(* CODESYS project Builder_Application_2RPi.project

Project tree, tasks and I/O mapping:
  Device : CODESYS Control for Raspberry Pi SL, 3S - Smart Software Solutions GmbH, version 3.5.11.0
    application Application
      libraries: Standard, * (System)
      task MainTask (cyclic, interval t#20ms, priority 1) calls PLC_PRG
      task VISU_TASK (cyclic, interval 100 ms, priority 31) calls VisuElems.Visu_Prg
      program PLC_PRG [ST]
      interface ITF_Builder: Set_Part1, Set_Part2, Set_Part3, Set_Main_Part
      function block ConcreteBuilder [ST]: Set_Main_Part, Set_Part1, Set_Part2, Set_Part3, Get_Main_Part, Get_Part1, Get_Part2, Get_Part3, Get_Result
      function block Director [ST]: fb_init, Construct
      function block Product [ST]: toString
      visualisation Visualization
    SoftMotion General Axis Pool
    GPIOs_A_B : GPIOs B+/Pi2, 3S - Smart Software Solutions GmbH, version 3.5.11.0
        unmapped channels: digital inputs (GPIO0..GPIO31), digital outputs (GPIO0..GPIO31)
    I²C
    SPI
    Onewire
    Camera device
      <Empty>
  libraries: VisuSymbols, 3.5.10.0 (System)
  text list GlobalTextList
*)

// Device/Application/PLC_PRG
PROGRAM PLC_PRG
VAR
	//Arrays with the different specifications for the Client to choose
	arrayChassis : ARRAY [1..3] OF STRING := ['Red Chassis ', 'Black Chassis ', 'White Chassis '];
	arrayCarType : ARRAY [1..3] OF STRING := ['Sedan ', 'Hatchback ', 'Sport '];
	arrayMotor : ARRAY [1..3] OF STRING := ['Motor 1.4cc ', 'Motor 2.0cc ', 'Motor 2.5cc '];
	arrayTires : ARRAY [1..3] OF STRING := ['Aluminium tires ', 'Chrome plated tires ', 'Ligth aluminium tires '];
	
	//Temporary array to have a reference to the clients choice
	tempArray : ARRAY [1..4] OF STRING;
	
	//Boolean and integer values to receive data from the tables in the visualization element
	//The boolean value validates if the client has chosen a valid option
	bChassis : BOOL := FALSE;
	//The integer value hold the reference to the array of specifications
	iChassis : INT := 0;
	
	//Boolean and integer values to receive data from the tables in the visualization element
	//The boolean value validates if the client has chosen a valid option
	bCarType : BOOL := FALSE;
	//The integer value hold the reference to the array of specifications
	iCarType : INT := 0;
	
	//Boolean and integer values to receive data from the tables in the visualization element
	//The boolean value validates if the client has chosen a valid option
	bMotor : BOOL := FALSE;
	//The integer value hold the reference to the array of specifications
	iMotor : INT := 0;
	
	//Boolean and integer values to receive data from the tables in the visualization element
	//The boolean value validates if the client has chosen a valid option
	bTires : BOOL := FALSE;
	//The integer value hold the reference to the array of specifications
	iTires : INT := 0;
	
	//Boolean value to verify and respond to a client's request
	bRequest : BOOL := FALSE;
	
	//String variable to interact and respond to the client in the visualization element
	sMessageLog : STRING := 'Waiting for your request';
	
	//A pointer to Poduct to dynamically create and delete product objects at the clients requests
	prod 	: POINTER TO Product;

	//A ConcreteBuilder instance to be passed to the Director and build the final Product objects
	aConcreteBuilder : ConcreteBuilder;
	
	//A Director instance that is instanciated with a ConcreteBuilder instance and the first specifications.
	// later on in the program these specifications of the ConcreteBuilder instance will be changed dynamically
	aDirector : Director(concreteBuilder:= aConcreteBuilder , specifications := tempArray);
	
END_VAR

//The visualization element has 4 coloums in which the client must select an option from each coloum.
//Once the client has made its choice, He can then procede to validate its request.
//The bottom rectangle will handle all possible responses from the application to the client.

//If the client makes a request in the visualization element
IF bRequest
	THEN
	//We verify that the cliet has chosen all the required parts(All in this case)
	IF bChassis AND bCarType AND bMotor AND bTires
		THEN
		//If the client has sent a valir request, the builder notifies the client about the received request
		sMessageLog := 'Your red car is being built';
		//A new product object is created on demand
		prod := __NEW(Product);
		//The tempArray is modified to the special characteristics demanded from the client on the visualization element
		tempArray[1] := arrayChassis[iChassis];
		tempArray[2] := arrayCarType[iCarType];
		tempArray[3] := arrayMotor[iMotor];
		tempArray[4] := arrayTires[iTires];

		//The Director object receives the specifications for the new Product to be built
		aDirector(spected := tempArray);
		//The Product object request the construction to the Director.
		prod^ := aDirector.Construct();
		//The Builder's response after the Director object has handled the proper request
		sMessageLog := CONCAT( 'Your car has been built. It has: ', prod^.toString());
		//Once this reques has been handled, the request flag is set to FALSE
		bRequest := FALSE;
		//Once this reques has been handled, the Product object is deleted to free memory
		__DELETE(prod);
		
		//If the client did not choose all the required parts
		ELSE
			
		//The Builder responds
		sMessageLog := 'You need to select all the parts for your car';
		//Once this reques has been handled, the reques flag is set to FALSE
		bRequest := FALSE;
		
	END_IF

END_IF

END_PROGRAM

// Device/Application/Product
{attribute 'enable_dynamic_creation'} 
//The class Product is just a plain blueprint of the components of the object to be built.
//The final Product may ot may not contain the all the Parts listed on the Product declaration
// rather only the parts in the specifications sent by the client.
FUNCTION_BLOCK Product
VAR_INPUT
	//List of possible parts to be build in a final Product object
	mainPart 	: STRING;
	part1 		: STRING;
	part2 		: STRING;
	part3 		: STRING;
END_VAR
VAR_OUTPUT
END_VAR
VAR
END_VAR

//Method to be used in the visualization element for an easier String handling
METHOD toString : STRING
VAR_INPUT
END_VAR

VAR
	//Local variable to join together and store the pieces of String
	tempString: STRING;
END_VAR
//tempString joins together "Main Part" and "Part 1" of the Product object
tempString := CONCAT(THIS^.mainPart , THIS^.part1);
//tempString joins together its current value and "Part 2" of the Product object
tempString := CONCAT(tempString , THIS^.part2);
//tempString joins together its current value and "Part 3" of the Product object
tempString := CONCAT(tempString , THIS^.part3);
//The final result is sent as the output of this method
toString := tempString;
END_METHOD

END_FUNCTION_BLOCK

// Device/Application/Director
//The director class is responsible to delegate the construction of the final product object 
// to a concrete builder object.
FUNCTION_BLOCK Director
VAR_INPUT
	//This variable is sent by the client as the specifications of the final product to be built.
	spected : ARRAY [1..4] OF STRING;
END_VAR
VAR_OUTPUT
END_VAR
VAR
	//Holds a reference to the concrete builder object to send the specifications of the final product to it.
	concreteBuilder : ConcreteBuilder;
	
	//Stores the specifications, sent by the client, of the final product to be built.
	specifications : ARRAY [1..4] OF STRING;
END_VAR

//This dynamic constructor changes the previous specifications of the final product to be built
THIS^.specifications := THIS^.spected;

//This constructor is called at instanciation to store the inital specifications of the product to be built and 
// the reference to the builder object.
METHOD fb_init
VAR_INPUT
	//Necesary fields for the constructor
	bInitRetains : BOOL; // TRUE: the Retain-variables are initialized (reset warm / reset cold)
	bInCopyCode : BOOL;  // TRUE  the instance will be copied to the copy-code afterward (online change)
	
	//Reference to the builder that is going to be building the final product object.
	concreteBuilder : ConcreteBuilder;	
	
	//Specifications, sent by the client, to be built on the final product object
	specifications : ARRAY [1..4] OF STRING;
	
END_VAR
//Stores the reference to which builder will be building the final product object in its own field THIS^.concreteBuilder
THIS^.concreteBuilder := concreteBuilder;

//Stores the specifications to build the final product object in its own field THIS^.specifications.
THIS^.specifications := specifications;
END_METHOD

//This method is going to be called by the client when a new Product object must be built
METHOD Construct : Product  
VAR_INPUT
END_VAR
//The Director tells its concreteBuilder instance to build the final product step by step passing the specifications stored in the 
// array THIS^.specifications[1..4]

//Step 1 "Main Part"
THIS^.concreteBuilder.Set_Main_Part(THIS^.specifications[1]);
//Step 2 "Part 1"
THIS^.concreteBuilder.Set_Part1(THIS^.specifications[2]);
//Step 3 "Part 2"
THIS^.concreteBuilder.Set_Part2(THIS^.specifications[3]);
//Step 4 "Part 3"
THIS^.concreteBuilder.Set_Part3(THIS^.specifications[4]);

//Finally the concreteBuilder instance in the Director object delivers the final result as a Product object
Construct := THIS^.concreteBuilder.Get_Result();
END_METHOD

END_FUNCTION_BLOCK

// Device/Application/ConcreteBuilder
//This is the concrete builder class, reponsible for building the final product object
FUNCTION_BLOCK ConcreteBuilder IMPLEMENTS ITF_Builder
VAR_INPUT
END_VAR
VAR_OUTPUT
END_VAR
VAR
	//Holds an internal reference to how the final product shoud be so the builder class can build it on the fly 
	// without any help from other classes exepting the Director class that is going to be passing the special
	//specifications to the builder.
	localProduct : Product;
END_VAR

//Illustrative method of the pattern to set the main part
METHOD Set_Main_Part
VAR_INPUT
	//Illustrative value (object because it is a TRING) to be set as a product part
	mainPart	: STRING;
END_VAR
//Sets the passed value to its corresponding field. 
//We can say that the the final product is in process of being built.
//So this is a step into building the final product done by the builder.
THIS^.localProduct.mainPart := mainPart;
END_METHOD

//Illustrative method of the pattern to set the part1
METHOD Set_Part1
VAR_INPUT
	//Illustrative value (object because it is a TRING) to be set as a product part
	part1	: STRING;
END_VAR
//Sets the passed value to its corresponding field. 
//We can say that the the final product is in process of being built.
//So this is a step into building the final product done by the builder.
THIS^.localProduct.part1 := part1;
END_METHOD

//Illustrative method of the pattern to set the part2
METHOD Set_Part2
VAR_INPUT
	//Illustrative value (object because it is a TRING) to be set as a product part
	part2	: STRING;
END_VAR
//Sets the passed value to its corresponding field. 
//We can say that the the final product is in process of being built.
//So this is a step into building the final product done by the builder.
THIS^.localProduct.part2 := part2;
END_METHOD

//Illustrative method of the pattern to set the part3
METHOD Set_Part3
VAR_INPUT
	//Illustrative value (object because it is a TRING) to be set as a product part
	part3	: STRING;
END_VAR
//Sets the passed value to its corresponding field. 
//We can say that the the final product is in process of being built.
//So this is a step into building the final product done by the builder.
THIS^.localProduct.part3 := part3;
END_METHOD

//Illustrative method of the pattern to get the main part
METHOD Get_Main_Part : STRING
VAR_INPUT
END_VAR
//Returns the object stored in the built product THIS^.localProduct.mainPart
Get_Main_Part := THIS^.localProduct.mainPart;
END_METHOD

//Illustrative method of the pattern to get the part1
METHOD Get_Part1 : STRING
VAR_INPUT
END_VAR
//Returns the object stored in the built product THIS^.localProduct.part1
Get_Part1 := THIS^.localProduct.part1;
END_METHOD

//Illustrative method of the pattern to get the part2
METHOD Get_Part2 : STRING
VAR_INPUT
END_VAR
//Returns the object stored in the built product THIS^.localProduct.part2
Get_Part2 := THIS^.localProduct.part2;
END_METHOD

//Illustrative method of the pattern to get the part3
METHOD Get_Part3 : STRING
VAR_INPUT
END_VAR
//Returns the object stored in the built product THIS^.localProduct.part3
Get_Part3 := THIS^.localProduct.part3;
END_METHOD

//Illustrative method of the pattern
METHOD Get_Result : Product
VAR_INPUT
END_VAR
VAR
END_VAR
//The concrete builder, after it builts the final object of class product, returns the 
// final product object 
Get_Result := THIS^.localProduct;
END_METHOD

END_FUNCTION_BLOCK

// Device/Application/ITF_Builder
//Builder interface to declare all needed parts to be built
INTERFACE ITF_Builder

//Illustrative method of the pattern to set the part1
METHOD Set_Part1
VAR_INPUT
	//Illustrative value (object because it is a TRING) to be set as a product part
	part1 : STRING;
END_VAR
END_METHOD

//Illustrative method of the pattern to set the part2
METHOD Set_Part2
VAR_INPUT
	//Illustrative value (object because it is a TRING) to be set as a product part
	part2 : String;
END_VAR
END_METHOD

//Illustrative method of the pattern to set the part3
METHOD Set_Part3
VAR_INPUT
	//Illustrative value (object because it is a TRING) to be set as a product part
	part3 : String;
END_VAR
END_METHOD

//Illustrative method of the pattern to set the main part
METHOD Set_Main_Part
VAR_INPUT
	//Illustrative value (object because it is a TRING) to be set as a product part
	mainPart : String;
END_VAR
END_METHOD

END_INTERFACE

// Device/Application/Visualization
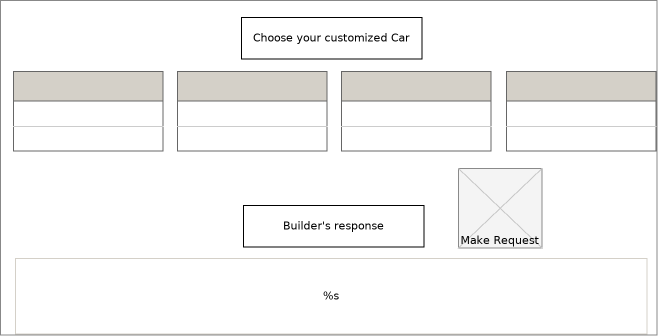
VISUALIZATION Visualization  // 658x336
//The visualization element has 4 coloums in which the client must select an option from each coloum.
//Once the client has made its choice, He can then procede to validate its request.
//The bottom rectangle will handle all possible responses from the application to the client.
    Table (13,71 150x80), data array: PLC_PRG.arrayChassis
        p3854506369: PLC_PRG.arrayChassis[INDEX]
        p2232123230: Chassis Colour
        p1137915858: PLC_PRG.iChassis
        p1822360349: PLC_PRG.bChassis
    Table (177,71 150x80), data array: PLC_PRG.arrayCarType
        p3854506369: PLC_PRG.arrayCarType[INDEX]
        p2232123230: Car Type
        p1137915858: PLC_PRG.iCarType
        p1822360349: PLC_PRG.bCarType
    Table (341,71 150x80), data array: PLC_PRG.arrayMotor
        p3854506369: PLC_PRG.arrayMotor[INDEX]
        p2232123230: Motor dimensions
        p1137915858: PLC_PRG.iMotor
        p1822360349: PLC_PRG.bMotor
    Table (506,71 150x80), data array: PLC_PRG.arrayTires
        p3854506369: PLC_PRG.arrayTires[INDEX]
        p1137915858: PLC_PRG.iTires
        p1822360349: PLC_PRG.bTires
    Image (458,168 84x80), "Make Request", image: VisuSymbols.Symbols.OK
        OnMouseClick:  ToggleVariable=PLC_PRG.bRequest
    Textfield (15,258 632x76), "%s", text variable: PLC_PRG.sMessageLog
    RoundedRectangle (241,17 181x42), "Choose your customized Car"
    RoundedRectangle (243,205 181x42), "Builder's response"
END_VISUALIZATION
